(* PLC project reAMsafe, BrAutomation SafeDESIGNER  5.16.0.0 *)
(* stored: companyURL http://www.br-automation.com, creationDateTime Thu Dec 05 14:10:31 2024 *)

PROGRAM Main

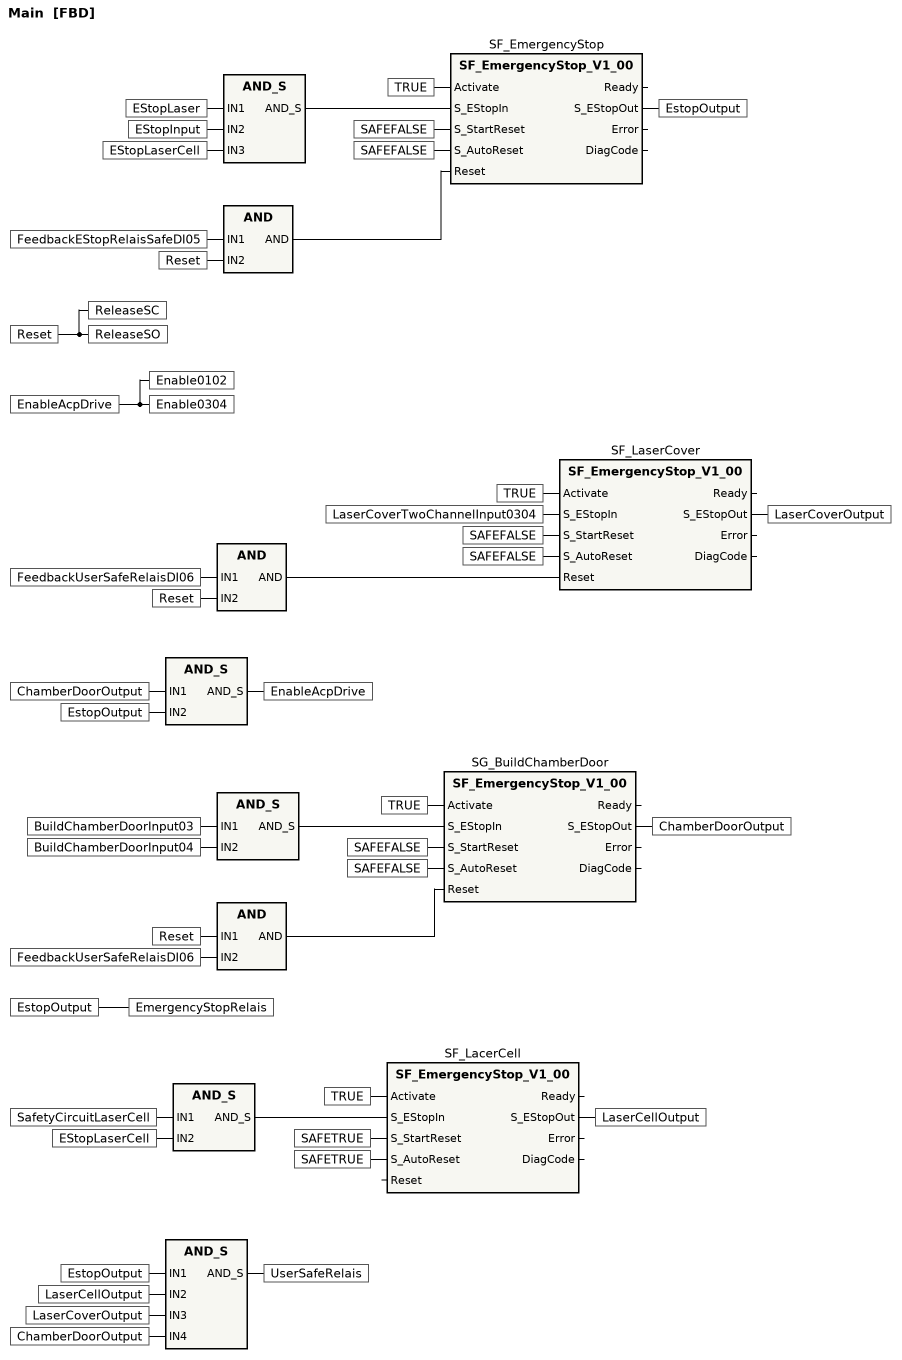
(* FBD diagram, written out as Structured Text *)
SF_LaserCover(Activate := TRUE, S_EStopIn := LaserCoverTwoChannelInput0304, S_StartReset := SAFEFALSE, S_AutoReset := SAFEFALSE, Reset := FeedbackUserSafeRelaisDI06 AND Reset);
LaserCoverOutput := SF_LaserCover.S_EStopOut;
SG_BuildChamberDoor(Activate := TRUE, S_EStopIn := AND_S(BuildChamberDoorInput03, BuildChamberDoorInput04), S_StartReset := SAFEFALSE, S_AutoReset := SAFEFALSE, Reset := Reset AND FeedbackUserSafeRelaisDI06);
ChamberDoorOutput := SG_BuildChamberDoor.S_EStopOut;
SF_EmergencyStop(Activate := TRUE, S_EStopIn := AND_S(EStopLaser, EStopInput, EStopLaserCell), S_StartReset := SAFEFALSE, S_AutoReset := SAFEFALSE, Reset := FeedbackEStopRelaisSafeDI05 AND Reset);
EstopOutput := SF_EmergencyStop.S_EStopOut;
SF_LacerCell(Activate := TRUE, S_EStopIn := AND_S(SafetyCircuitLaserCell, EStopLaserCell), S_StartReset := SAFETRUE, S_AutoReset := SAFETRUE);
LaserCellOutput := SF_LacerCell.S_EStopOut;
EnableAcpDrive := AND_S(ChamberDoorOutput, EstopOutput);
UserSafeRelais := AND_S(EstopOutput, LaserCellOutput, LaserCoverOutput, ChamberDoorOutput);
Enable0304 := EnableAcpDrive;
Enable0102 := EnableAcpDrive;
EmergencyStopRelais := EstopOutput;
ReleaseSO := Reset;
ReleaseSC := Reset;
END_PROGRAM
